(* PLC project faults, TNI-Software ControlBuild 4.00.17 *)
(* stored: creationDateTime 2005-06-20T11:52:29-01:00 *)

FUNCTION_BLOCK cmd_equipment_library.faults
  VAR_INPUT  (* CB.group=Orders CB.kind=inputVars *)
    forwardCmd : BOOL := false;  (* CB.libelle=Forward command *)
  END_VAR
  VAR_INPUT  (* CB.group=FeedBacks CB.kind=inputVars *)
    thermalFB : BOOL := false;  (* CB.mnemonicPatternPropertyName=<SY>_THER_<NU> CB.libelle=Feedback of the thermal protection of the engine *)
    forwardFB : BOOL := false;  (* CB.libelle=Forward feedback *)
  END_VAR
  VAR_INPUT  (* CB.kind=inputVars *)
    acknowledgePB : BOOL := false;  (* CB.mnemonicPatternPropertyName=<SY>_PBACK_<NU> CB.libelle=Acknowledgement pushbutton *)
  END_VAR
  VAR_OUTPUT  (* CB.kind=outputVars *)
    generalFault : BOOL := false;  (* CB.mnemonicPatternPropertyName=grlFlt<SY><NU> CB.libelle=General fault of the engine *)
  END_VAR
  VAR CONSTANT  (* CB.kind=parameterVars *)
    preset : DINT := 2;  (* CB.mnemonicPatternPropertyName=preset<SY><NU> *)
  END_VAR
  VAR  (* CB.group=Faults CB.kind=overControlVars *)
    thermalFault : BOOL := false;  (* CB.mnemonicPatternPropertyName=thermalFlt<SY><NU> CB.libelle=Thermal (electric) fault *)
    forwardFault : BOOL := false;  (* CB.mnemonicPatternPropertyName=fwdFlt<SY><NU> CB.libelle=Fault of the forward feedback *)
  END_VAR

(* LD diagram, written out as Structured Text *)
1:
IF acknowledgePB THEN thermalFault := FALSE; END_IF;
IF acknowledgePB THEN forwardFault := FALSE; END_IF;
IF acknowledgePB THEN generalFault := FALSE; END_IF;
2:
ton_sec_1(IN := forwardCmd, PT := preset);
IF ton_sec_1.Q AND NOT forwardFB THEN forwardFault := TRUE; END_IF;
3:
ton_sec_2(IN := NOT thermalFB, PT := preset);
IF ton_sec_2.Q THEN thermalFault := TRUE; END_IF;
4:
IF forwardFault OR thermalFault THEN generalFault := TRUE; END_IF;
END_FUNCTION_BLOCK
